(* Logix 5000 project; controller Hose_HP_Test_Rig_V1 vendor 1 type 14 code 149 rev 32.11; software revision 32.00; part 3 of 10 *)
(* tags used below, declared in another part *)
   DOOR_CLOSE_STS_STN1 : DINT;
   EXHS_OK_DEL_STN1 : TIMER;
   EXHS_VAL_OFF_CE_STN1 : BOOL;
   EXHS_VAL_OFF_TE_STN1 : BOOL;
   ONS26 : BOOL;
   ONS27 : BOOL;
   ONS43 : BOOL;
   ONS44 : BOOL;
   ONS45 : BOOL;
   ONS71 : BOOL;
   ONS72 : BOOL;
   ONS73 : BOOL;
   ONS74 : BOOL;
   ONS75 : BOOL;
   PASS_COUNTER_STN1 : COUNTER;
   PASS_COUNTER_STN2 : COUNTER;
   PASS_COUNTER_STN3 : COUNTER;
   PASS_COUNTER_STN4 : COUNTER;
   RST_TOP_NOT_DECLAMPED_STN1 : BOOL;
   RST_TOP_NOT_DECLAMPED_STN2 : BOOL;
   RST_TOP_NOT_DECLAMPED_STN3 : BOOL;
   RST_TOP_NOT_DECLAMPED_STN4 : BOOL;
   ABORT_STN1 : BOOL;
   ACT_DROP_STN1 : REAL;
   ACT_PR_STN1 : REAL;
   AUTO_DOOR_OPEN_BLK_STN1 : DA_SOL_RET_SEQ;
   AUTO_DOOR_OPEN_BLK_STN2 : DA_SOL_RET_SEQ;
   AUTO_DOOR_OPEN_BLK_STN3 : DA_SOL_RET_SEQ;
   AUTO_DOOR_OPEN_BLK_STN4 : DA_SOL_RET_SEQ;
   AUTO_DOOR_OPEN_ON : BOOL;
   AUTO_DOOR_OPEN_ON_STN2 : BOOL;
   AUTO_DOOR_OPEN_ON_STN3 : BOOL;
   AUTO_DOOR_OPEN_ON_STN4 : BOOL;
   AUTO_DOOR_OPEN_SEQ : DINT;
   AUTO_DOOR_OPEN_SEQ_STN2 : DINT;
   AUTO_DOOR_OPEN_SEQ_STN3 : DINT;
   AUTO_DOOR_OPEN_SEQ_STN4 : DINT;
   AUTO_TEST_ON_STN1 : BOOL;
   AUTO_TEST_ON_STN2 : BOOL;
   AUTO_TEST_ON_STN3 : BOOL;
   AUTO_TEST_ON_STN4 : BOOL;
   AUTO_TEST_OVER_STN1 : BOOL;
   AUTO_TEST_OVER_STN2 : BOOL;
   AUTO_TEST_OVER_STN3 : BOOL;
   AUTO_TEST_OVER_STN4 : BOOL;
   AUTO_TEST_SEL_STN1 : BOOL;
   AUTO_TEST_SEL_STN2 : BOOL;
   AUTO_TEST_SEL_STN3 : BOOL;
   AUTO_TEST_SEL_STN4 : BOOL;
   BOTTOM_CLAMP_AUTO_STN1 : BOOL;
   BOTTOM_CLAMP_BLK_STN1 : DA_SOL_FWD_SEQ;
   BOTTOM_CLAMP_OK_STN1 : BOOL;
   BOTTOM_CLAMP_PR_CHK : TIMER;
   BOTTOM_CLAMP_PS_STN1 : ALIAS FOR Local:1:I.Data.13;
   BOTTOM_CLAMP_PS_STN2 : ALIAS FOR Local:2:I.Data.2;
   BOTTOM_CLAMP_PS_STN3 : ALIAS FOR Local:2:I.Data.7;
   BOTTOM_CLAMP_PS_STN4 : ALIAS FOR Local:2:I.Data.12;
   BOTTOM_CLAMP_SEQ_STN1 : DINT;
   BOTTOM_CLAMP_SOL_STN1 : ALIAS FOR Local:1:O.Data.4;
   BOTTOM_DECLAMP_AUTO_STN1 : BOOL;
   BOTTOM_DECLAMP_SEQ_STN1 : DINT;
   BOTTOM_DECLMP_BLK_STN1 : DA_SOL_RET_SEQ;
   BOTTOM_NOT_CLAMPED_STN1 : BOOL;
   BOTTOM_NOT_DECLAMPED_STN1 : BOOL;
   CHECK_TRACE_STS_STN1 : BOOL;
   CLR_FAIL_ONS_STN1 : BOOL;
   CLR_ONS_STN1 : BOOL;
   COMP_FAULT_STN1 : BOOL;
   CONS_CALB_OFF_STN1 : BOOL;
   CONS_CALB_OFF_STN2 : BOOL;
   CONS_CALB_OFF_STN3 : BOOL;
   CONS_CALB_OFF_STN4 : BOOL;
   CONS_CALB_ON_STN1 : BOOL;
   CONS_STS_STN1 : DINT;
   CONS_TEST_ON : BOOL;
   CONSTRICTION_TEST_ON_STN1 : BOOL;
   CONSTRICTION_TEST_ON_STN2 : BOOL;
   CONSTRICTION_TEST_ON_STN3 : BOOL;
   CONSTRICTION_TEST_ON_STN4 : BOOL;
   DICH_STN1 : INT;
   DOOR_CLOSE_ABORT_STN1 : BOOL;
   DOOR_CLOSE_AUTO_STN1 : BOOL;
   DOOR_CLOSE_BLK_STN1 : DOOR_CLOSE;
   DOOR_CLOSE_OK_STN1 : BOOL;
   DOOR_CLOSE_RS_STN1 : ALIAS FOR Local:1:I.Data.11;
   DOOR_CLOSE_SEQ_STN1 : DA_SOL_FWD_SEQ;
   DOOR_NOT_CLOSED : BOOL;
   DOOR_NOT_OPEN_STN1 : BOOL;
   DOOR_NOT_OPEN_STN2 : BOOL;
   DOOR_NOT_OPEN_STN3 : BOOL;
   DOOR_NOT_OPEN_STN4 : BOOL;
   DOOR_OPEN_RS_STN1 : ALIAS FOR Local:1:I.Data.10;
   DOOR_OPEN_RS_STN2 : ALIAS FOR Local:1:I.Data.15;
   DOOR_OPEN_RS_STN3 : ALIAS FOR Local:2:I.Data.4;
   DOOR_OPEN_RS_STN4 : ALIAS FOR Local:2:I.Data.10;
   DROP_CHK_SEQ_STN1 : DROP_CHECK;
   DROP_NOK_STN1 : BOOL;
   DROP_OK_STN1 : BOOL;
   DUPLICATE_STN1 : BOOL;
   EC_STN1 : DINT;
   EC_STN2 : DINT;
   EC_STN3 : DINT;
   EC_STN4 : DINT;
   EXHAUST_SET_LIM : REAL;
   EXHS_OFF_BLK_STN1 : FILL_VAL_OFF;
   EXHS_VAL_HP_ON_STN1 : BOOL;
   EXHS_VAL_OFF_STN1 : BOOL;
   FAILED_STN1 : BOOL;
   FAILED_STN2 : BOOL;
   FAILED_STN3 : BOOL;
   FAILED_STN4 : BOOL;
   FAULTED_STN1 : BOOL;
   FAULTED_STN2 : BOOL;
   FAULTED_STN3 : BOOL;
   FAULTED_STN4 : BOOL;
   FILL_ACT_TIME_STN1 : REAL;
   FILL_CHK_STN1 : PR_CHECK;
   FILL_HIGH_STN1 : BOOL;
   FILL_HL_STN1 : REAL;
   FILL_LL_STN1 : REAL;
   FILL_LOW_STN1 : BOOL;
   FILL_SEQ_START_STN : SEQ_START_AND_FILL;
   FILL_SET_TIME : REAL;
   FILL_VAL_OFF_SEQ_STN1 : FILL_VAL_OFF;
   FLT_CLR_ONS_STN1 : BOOL;
   FLT_CLR_ONS_STN2 : BOOL;
   FLT_CLR_ONS_STN3 : BOOL;
   FLT_CLR_ONS_STN4 : BOOL;
   FLT_CODE_STN4 : DINT;
   HP_P2_STN1 : REAL;
   HP_STS_STN1 : DINT;
   HP_TEST_ON : BOOL;
   INCORRECT_STN1 : BOOL;
   INIT_STN1 : BOOL;
   LT_COMPLETED_STN1 : BOOL;
   LT_P1_STN1 : REAL;
   LT_POKEYOKE_STN1 : DINT;
   MSG_STN1 : DINT;
   MSG_STN2 : DINT;
   MSG_STN3 : DINT;
   MSG_STN4 : DINT;
   P2_STN1 : REAL;
   PASS_COUNT_RETEST : DINT;
   PASS_COUNT_RETEST_STN2 : DINT;
   PASS_COUNT_STN1 : DINT;
   PASS_COUNT_STN2 : DINT;
   PASS_COUNT_STN3 : DINT;
   PASS_COUNT_STN4 : DINT;
   PASS_COUNTER_RETEST : COUNTER;
   PASS_COUNTER_RETEST_STN2 : COUNTER;
   PASSED_STN1 : BOOL;
   PASSED_STN2 : BOOL;
   PASSED_STN3 : BOOL;
   PASSED_STN4 : BOOL;
   POKEYOKE_NOT_DONE : BOOL;
   PYOKE_LT_STN1 : BOOL;
   RETEST : BOOL;
   RST_EXHS_VAL_OFF_STN1 : BOOL;
   RST_SEQ_ON_STN1 : BOOL;
   RST_TEST_VAL_OFF_STN1 : BOOL;
   SCAN_OK_STN1 : BOOL;
   SCR_STS : DINT[6];
   SEQ_NO_STN1 : DINT;
   SEQ_NO_STN2 : DINT;
   SEQ_NO_STN3 : DINT;
   SEQ_NO_STN4 : DINT;
   SET_DROP : REAL;
   STAB_ACT_TIME_STN1 : REAL;
   STAB_CHK_STN1 : PR_CHECK;
   STAB_HIGH_STN1 : BOOL;
   STAB_LOW_STN1 : BOOL;
   STAB_SET_TIME : REAL;
   STAMP_BLK_STN1 : STAMP_SEQ;
   STAMP_BLK_STN2 : STAMP_SEQ;
   STAMP_BLK_STN3 : STAMP_SEQ;
   STAMP_BLK_STN4 : STAMP_SEQ;
   STAMP_FWD_OK_STN1 : BOOL;
   STAMP_FWD_OK_STN2 : BOOL;
   STAMP_FWD_OK_STN3 : BOOL;
   STAMP_FWD_OK_STN4 : BOOL;
   STAMP_NOT_FWD : BOOL;
   STAMP_NOT_FWD_STN2 : BOOL;
   STAMP_NOT_FWD_STN3 : BOOL;
   STAMP_NOT_FWD_STN4 : BOOL;
   STAMP_ON_STN1 : BOOL;
   STAMP_ON_STN2 : BOOL;
   STAMP_ON_STN3 : BOOL;
   STAMP_ON_STN4 : BOOL;
   STAMP_PS_STN1 : ALIAS FOR Local:1:I.Data.14;
   STAMP_PS_STN2 : ALIAS FOR Local:2:I.Data.3;
   STAMP_PS_STN3 : ALIAS FOR Local:2:I.Data.8;
   STAMP_PS_STN4 : ALIAS FOR Local:2:I.Data.13;
   STN1_ON : BOOL;
   STN1_TEST_STS : DINT;
   STN2_TEST_STS : DINT;
   STN3_TEST_STS : DINT;
   STN4_TEST_STS : DINT;
   STS_OP_STN1 : DINT;
   TEST_ACT_TIME_STN1 : REAL;
   TEST_ON_STN1 : BOOL;
   TEST_ON_STN2 : BOOL;
   TEST_ON_STN3 : BOOL;
   TEST_ON_STN4 : BOOL;
   TEST_OVER_DEL : TIMER;
   TEST_OVER_DEL_STN2 : TIMER;
   TEST_OVER_DEL_STN3 : TIMER;
   TEST_OVER_DEL_STN4 : TIMER;
   TEST_SET_TIME : REAL;
   TEST_STS_STN1 : DINT;
   TEST_STS_UPDATE_STN1 : TEST_TAIL_END;
   TEST_VAL_OFF_STN1 : BOOL;
   TEST_VAL_ON_STN1 : BOOL;
   TOP_CLAMP_AUTO_STN1 : BOOL;
   TOP_CLAMP_BLK_STN1 : DA_SOL_FWD_SEQ;
   TOP_CLAMP_OK_STN1 : BOOL;
   TOP_CLAMP_ON_SEQ_STN1 : DINT;
   TOP_CLAMP_PS_STN1 : ALIAS FOR Local:1:I.Data.12;
   TOP_CLAMP_PS_STN2 : ALIAS FOR Local:2:I.Data.1;
   TOP_CLAMP_PS_STN3 : ALIAS FOR Local:2:I.Data.6;
   TOP_CLAMP_PS_STN4 : ALIAS FOR Local:2:I.Data.11;
   TOP_DECLAMP_AUTO_STN1 : BOOL;
   TOP_DECLAMP_AUTO_STN2 : BOOL;
   TOP_DECLAMP_AUTO_STN3 : BOOL;
   TOP_DECLAMP_AUTO_STN4 : BOOL;
   TOP_DECLAMP_BLK_STN1 : TOP_DECLAMP;
   TOP_DECLAMP_BLK_STN2 : TOP_DECLAMP;
   TOP_DECLAMP_BLK_STN3 : TOP_DECLAMP;
   TOP_DECLAMP_BLK_STN4 : TOP_DECLAMP;
   TOP_DECLAMP_OK_STN1 : BOOL;
   TOP_DECLAMP_OK_STN2 : BOOL;
   TOP_DECLAMP_OK_STN3 : BOOL;
   TOP_DECLAMP_OK_STN4 : BOOL;
   TOP_NOT_CLAMPED_STN1 : BOOL;
   TOP_NOT_DECLAMPED_STN1 : BOOL;
   TOP_NOT_DECLAMPED_STN2 : BOOL;
   TOP_NOT_DECLAMPED_STN3 : BOOL;
   TOP_NOT_DECLAMPED_STN4 : BOOL;
   TRACE_ON_STN1 : BOOL;
   TS_STS_OP20A : DINT;
   TS_STS_STN1 : DINT;
   TS_STS_STN3 : DINT;
   TS_STS_STN4 : DINT;
(* MainProgram, continued *)

ROUTINE Auto_End_Stn1   (* ladder *)
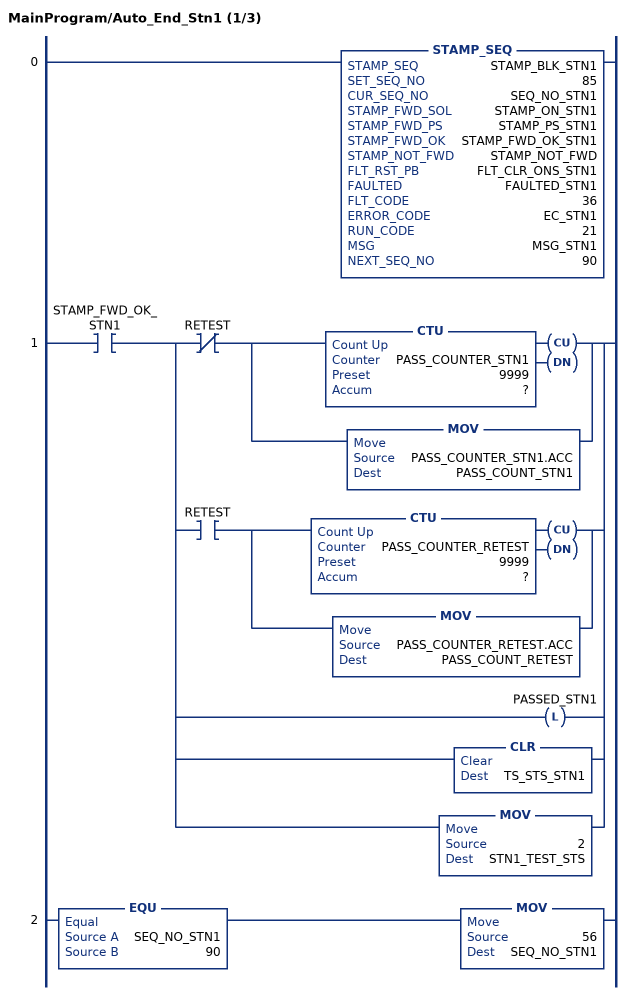
   0: STAMP_SEQ(STAMP_BLK_STN1,85,SEQ_NO_STN1,STAMP_ON_STN1,STAMP_PS_STN1,STAMP_FWD_OK_STN1,STAMP_NOT_FWD,FLT_CLR_ONS_STN1,FAULTED_STN1,36,EC_STN1,21,MSG_STN1,90);
   1: XIC(STAMP_FWD_OK_STN1)[XIO(RETEST) [CTU(PASS_COUNTER_STN1,?,?) ,MOV(PASS_COUNTER_STN1.ACC,PASS_COUNT_STN1) ] ,XIC(RETEST) [CTU(PASS_COUNTER_RETEST,?,?) ,MOV(PASS_COUNTER_RETEST.ACC,PASS_COUNT_RETEST) ] ,OTL(PASSED_STN1) ,CLR(TS_STS_STN1) ,MOV(2,STN1_TEST_STS) ];
   2: EQU(SEQ_NO_STN1,90)MOV(56,SEQ_NO_STN1);
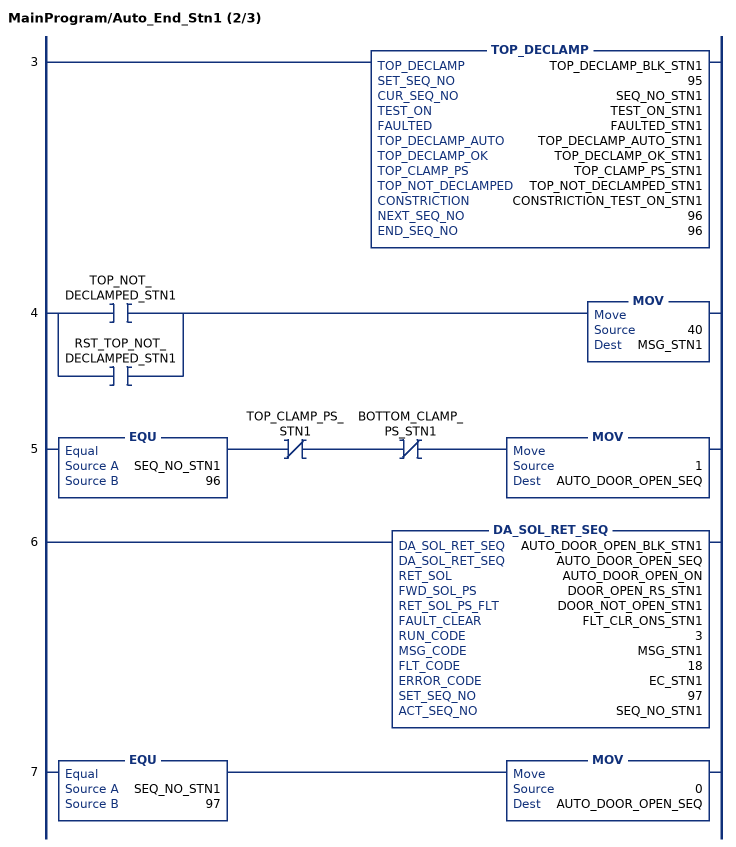
   3: TOP_DECLAMP(TOP_DECLAMP_BLK_STN1,95,SEQ_NO_STN1,TEST_ON_STN1,FAULTED_STN1,TOP_DECLAMP_AUTO_STN1,TOP_DECLAMP_OK_STN1,TOP_CLAMP_PS_STN1,TOP_NOT_DECLAMPED_STN1,CONSTRICTION_TEST_ON_STN1,96,96);
   4: [XIC(TOP_NOT_DECLAMPED_STN1) ,XIC(RST_TOP_NOT_DECLAMPED_STN1) ]MOV(40,MSG_STN1);
   5: EQU(SEQ_NO_STN1,96)XIO(TOP_CLAMP_PS_STN1)XIO(BOTTOM_CLAMP_PS_STN1)MOV(1,AUTO_DOOR_OPEN_SEQ);
   6: DA_SOL_RET_SEQ(AUTO_DOOR_OPEN_BLK_STN1,AUTO_DOOR_OPEN_SEQ,AUTO_DOOR_OPEN_ON,DOOR_OPEN_RS_STN1,DOOR_NOT_OPEN_STN1,FLT_CLR_ONS_STN1,3,MSG_STN1,18,EC_STN1,97,SEQ_NO_STN1);
   7: EQU(SEQ_NO_STN1,97)MOV(0,AUTO_DOOR_OPEN_SEQ);
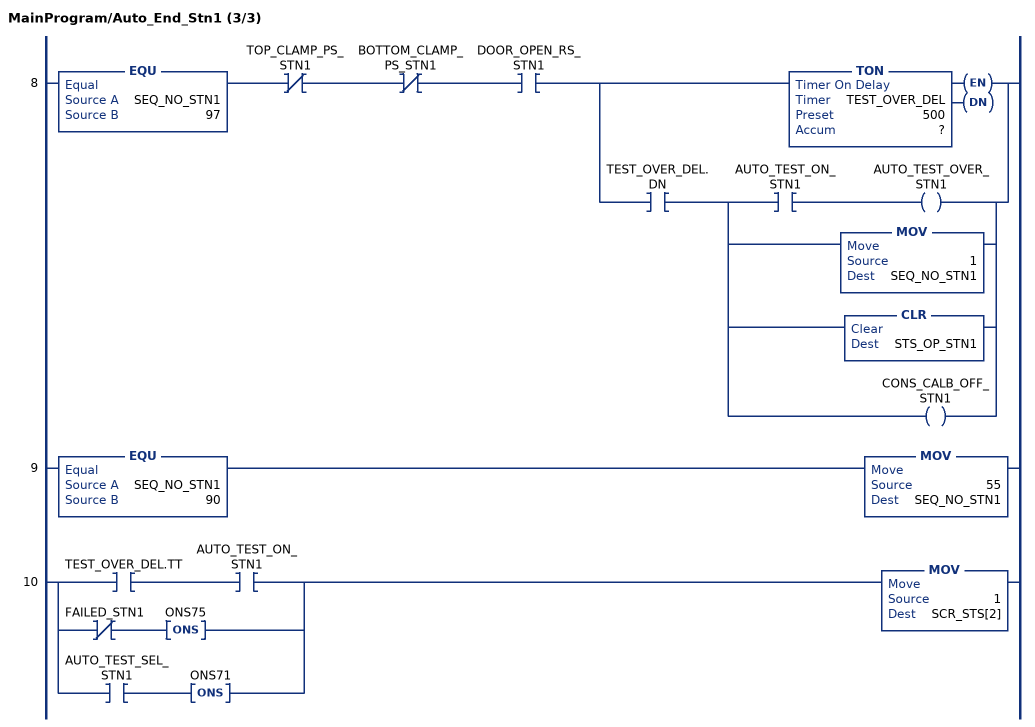
   8: EQU(SEQ_NO_STN1,97)XIO(TOP_CLAMP_PS_STN1)XIO(BOTTOM_CLAMP_PS_STN1)XIC(DOOR_OPEN_RS_STN1)[TON(TEST_OVER_DEL,?,?) ,XIC(TEST_OVER_DEL.DN) [[XIC(AUTO_TEST_ON_STN1) OTE(AUTO_TEST_OVER_STN1) ,MOV(1,SEQ_NO_STN1) ,CLR(STS_OP_STN1) ] ,OTE(CONS_CALB_OFF_STN1) ] ];
   9: EQU(SEQ_NO_STN1,90)MOV(55,SEQ_NO_STN1);
   10: [XIC(TEST_OVER_DEL.TT) XIC(AUTO_TEST_ON_STN1) ,XIO(FAILED_STN1) ONS(ONS75) ,XIC(AUTO_TEST_SEL_STN1) ONS(ONS71) ]MOV(1,SCR_STS[2]);
END_ROUTINE

ROUTINE Auto_End_Stn2   (* ladder *)
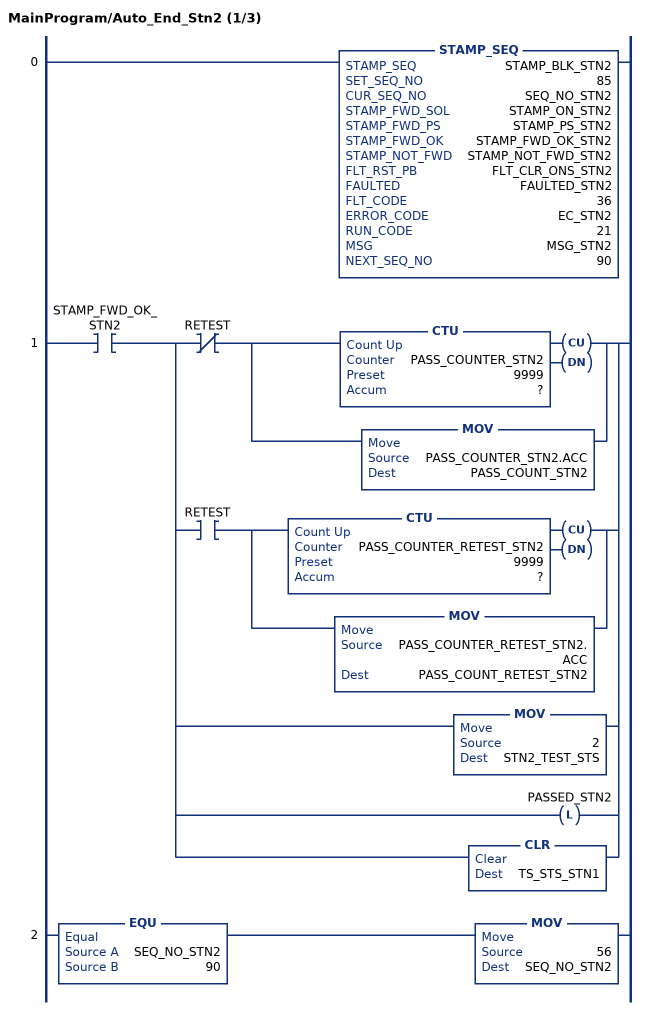
   0: STAMP_SEQ(STAMP_BLK_STN2,85,SEQ_NO_STN2,STAMP_ON_STN2,STAMP_PS_STN2,STAMP_FWD_OK_STN2,STAMP_NOT_FWD_STN2,FLT_CLR_ONS_STN2,FAULTED_STN2,36,EC_STN2,21,MSG_STN2,90);
   1: XIC(STAMP_FWD_OK_STN2)[XIO(RETEST) [CTU(PASS_COUNTER_STN2,?,?) ,MOV(PASS_COUNTER_STN2.ACC,PASS_COUNT_STN2) ] ,XIC(RETEST) [CTU(PASS_COUNTER_RETEST_STN2,?,?) ,MOV(PASS_COUNTER_RETEST_STN2.ACC,PASS_COUNT_RETEST_STN2) ] ,MOV(2,STN2_TEST_STS) ,OTL(PASSED_STN2) ,CLR(TS_STS_STN1) ];
   2: EQU(SEQ_NO_STN2,90)MOV(56,SEQ_NO_STN2);
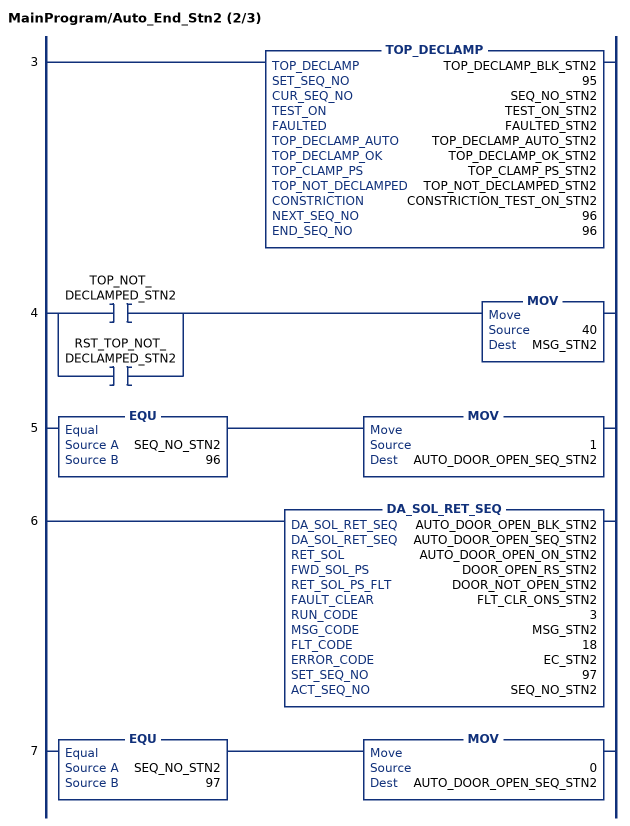
   3: TOP_DECLAMP(TOP_DECLAMP_BLK_STN2,95,SEQ_NO_STN2,TEST_ON_STN2,FAULTED_STN2,TOP_DECLAMP_AUTO_STN2,TOP_DECLAMP_OK_STN2,TOP_CLAMP_PS_STN2,TOP_NOT_DECLAMPED_STN2,CONSTRICTION_TEST_ON_STN2,96,96);
   4: [XIC(TOP_NOT_DECLAMPED_STN2) ,XIC(RST_TOP_NOT_DECLAMPED_STN2) ]MOV(40,MSG_STN2);
   5: EQU(SEQ_NO_STN2,96)MOV(1,AUTO_DOOR_OPEN_SEQ_STN2);
   6: DA_SOL_RET_SEQ(AUTO_DOOR_OPEN_BLK_STN2,AUTO_DOOR_OPEN_SEQ_STN2,AUTO_DOOR_OPEN_ON_STN2,DOOR_OPEN_RS_STN2,DOOR_NOT_OPEN_STN2,FLT_CLR_ONS_STN2,3,MSG_STN2,18,EC_STN2,97,SEQ_NO_STN2);
   7: EQU(SEQ_NO_STN2,97)MOV(0,AUTO_DOOR_OPEN_SEQ_STN2);
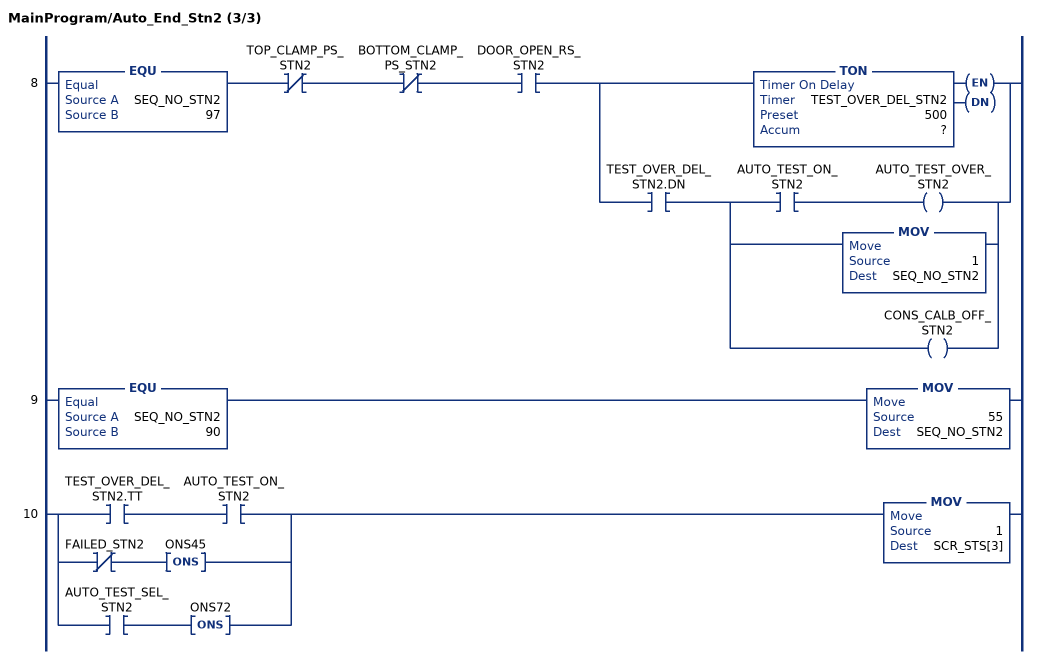
   8: EQU(SEQ_NO_STN2,97)XIO(TOP_CLAMP_PS_STN2)XIO(BOTTOM_CLAMP_PS_STN2)XIC(DOOR_OPEN_RS_STN2)[TON(TEST_OVER_DEL_STN2,?,?) ,XIC(TEST_OVER_DEL_STN2.DN) [XIC(AUTO_TEST_ON_STN2) OTE(AUTO_TEST_OVER_STN2) ,MOV(1,SEQ_NO_STN2) ,OTE(CONS_CALB_OFF_STN2) ] ];
   9: EQU(SEQ_NO_STN2,90)MOV(55,SEQ_NO_STN2);
   10: [XIC(TEST_OVER_DEL_STN2.TT) XIC(AUTO_TEST_ON_STN2) ,XIO(FAILED_STN2) ONS(ONS45) ,XIC(AUTO_TEST_SEL_STN2) ONS(ONS72) ]MOV(1,SCR_STS[3]);
END_ROUTINE

ROUTINE Auto_End_Stn3   (* ladder *)
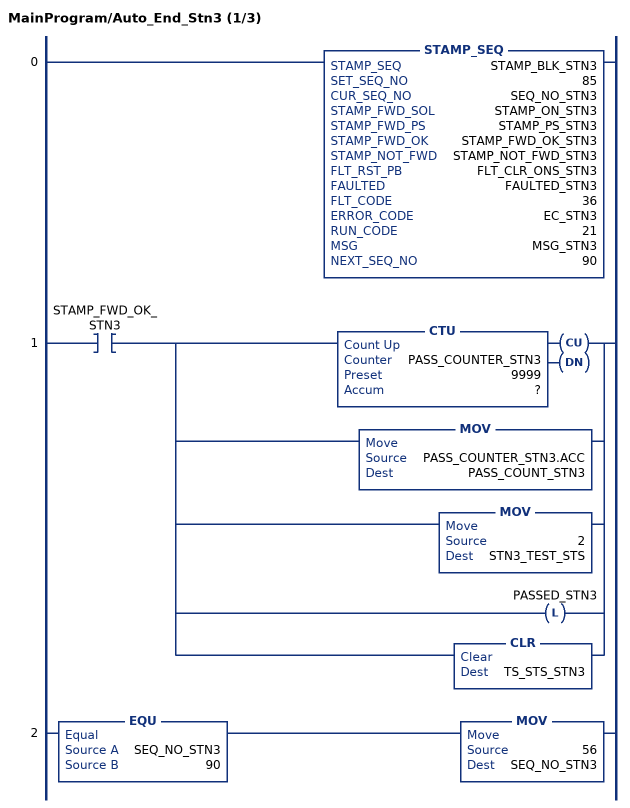
   0: STAMP_SEQ(STAMP_BLK_STN3,85,SEQ_NO_STN3,STAMP_ON_STN3,STAMP_PS_STN3,STAMP_FWD_OK_STN3,STAMP_NOT_FWD_STN3,FLT_CLR_ONS_STN3,FAULTED_STN3,36,EC_STN3,21,MSG_STN3,90);
   1: XIC(STAMP_FWD_OK_STN3)[CTU(PASS_COUNTER_STN3,?,?) ,MOV(PASS_COUNTER_STN3.ACC,PASS_COUNT_STN3) ,MOV(2,STN3_TEST_STS) ,OTL(PASSED_STN3) ,CLR(TS_STS_STN3) ];
   2: EQU(SEQ_NO_STN3,90)MOV(56,SEQ_NO_STN3);
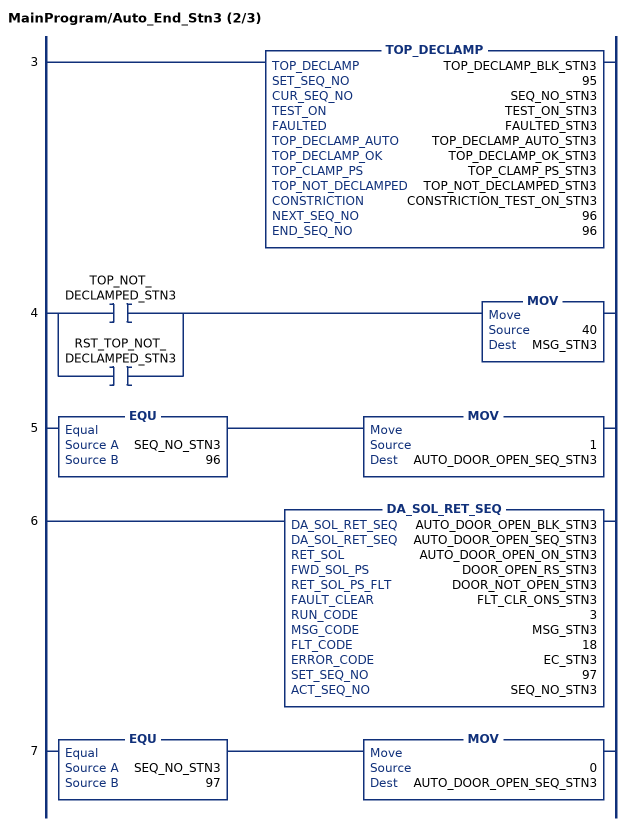
   3: TOP_DECLAMP(TOP_DECLAMP_BLK_STN3,95,SEQ_NO_STN3,TEST_ON_STN3,FAULTED_STN3,TOP_DECLAMP_AUTO_STN3,TOP_DECLAMP_OK_STN3,TOP_CLAMP_PS_STN3,TOP_NOT_DECLAMPED_STN3,CONSTRICTION_TEST_ON_STN3,96,96);
   4: [XIC(TOP_NOT_DECLAMPED_STN3) ,XIC(RST_TOP_NOT_DECLAMPED_STN3) ]MOV(40,MSG_STN3);
   5: EQU(SEQ_NO_STN3,96)MOV(1,AUTO_DOOR_OPEN_SEQ_STN3);
   6: DA_SOL_RET_SEQ(AUTO_DOOR_OPEN_BLK_STN3,AUTO_DOOR_OPEN_SEQ_STN3,AUTO_DOOR_OPEN_ON_STN3,DOOR_OPEN_RS_STN3,DOOR_NOT_OPEN_STN3,FLT_CLR_ONS_STN3,3,MSG_STN3,18,EC_STN3,97,SEQ_NO_STN3);
   7: EQU(SEQ_NO_STN3,97)MOV(0,AUTO_DOOR_OPEN_SEQ_STN3);
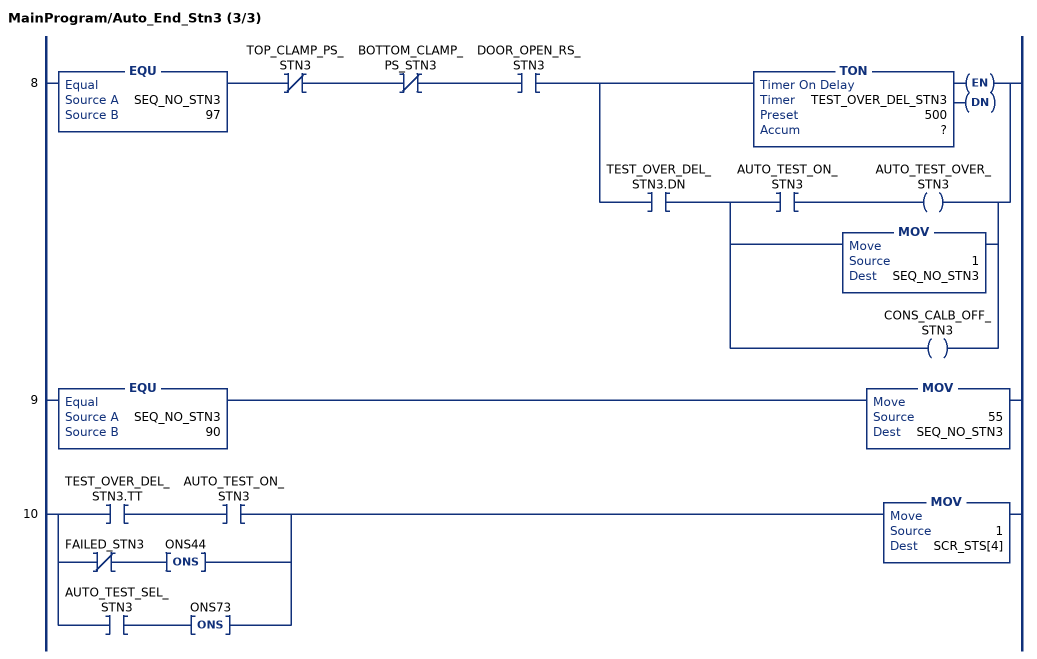
   8: EQU(SEQ_NO_STN3,97)XIO(TOP_CLAMP_PS_STN3)XIO(BOTTOM_CLAMP_PS_STN3)XIC(DOOR_OPEN_RS_STN3)[TON(TEST_OVER_DEL_STN3,?,?) ,XIC(TEST_OVER_DEL_STN3.DN) [XIC(AUTO_TEST_ON_STN3) OTE(AUTO_TEST_OVER_STN3) ,MOV(1,SEQ_NO_STN3) ,OTE(CONS_CALB_OFF_STN3) ] ];
   9: EQU(SEQ_NO_STN3,90)MOV(55,SEQ_NO_STN3);
   10: [XIC(TEST_OVER_DEL_STN3.TT) XIC(AUTO_TEST_ON_STN3) ,XIO(FAILED_STN3) ONS(ONS44) ,XIC(AUTO_TEST_SEL_STN3) ONS(ONS73) ]MOV(1,SCR_STS[4]);
END_ROUTINE

ROUTINE Auto_End_Stn4   (* ladder *)
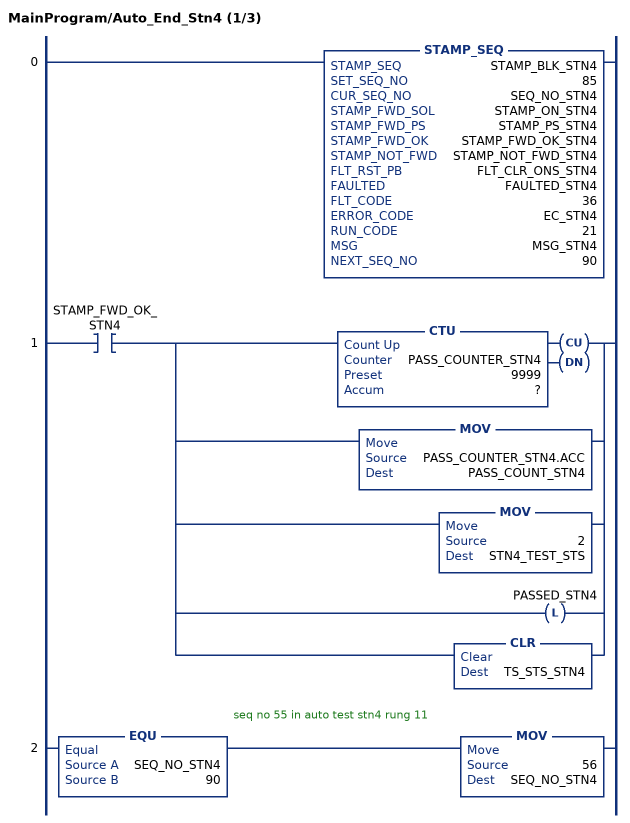
   0: STAMP_SEQ(STAMP_BLK_STN4,85,SEQ_NO_STN4,STAMP_ON_STN4,STAMP_PS_STN4,STAMP_FWD_OK_STN4,STAMP_NOT_FWD_STN4,FLT_CLR_ONS_STN4,FAULTED_STN4,36,EC_STN4,21,MSG_STN4,90);
   1: XIC(STAMP_FWD_OK_STN4)[CTU(PASS_COUNTER_STN4,?,?) ,MOV(PASS_COUNTER_STN4.ACC,PASS_COUNT_STN4) ,MOV(2,STN4_TEST_STS) ,OTL(PASSED_STN4) ,CLR(TS_STS_STN4) ];
   // seq no 55 in auto test stn4 rung 11
   2: EQU(SEQ_NO_STN4,90)MOV(56,SEQ_NO_STN4);
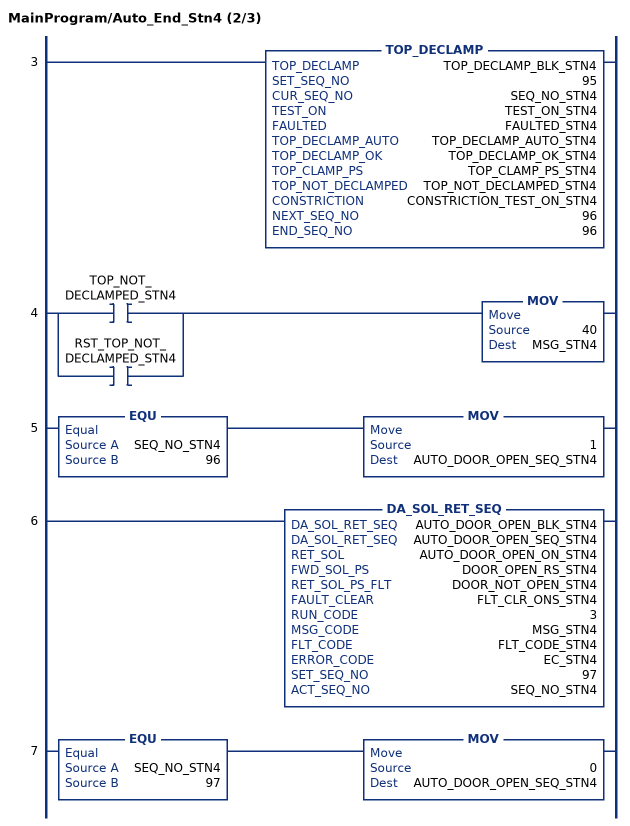
   3: TOP_DECLAMP(TOP_DECLAMP_BLK_STN4,95,SEQ_NO_STN4,TEST_ON_STN4,FAULTED_STN4,TOP_DECLAMP_AUTO_STN4,TOP_DECLAMP_OK_STN4,TOP_CLAMP_PS_STN4,TOP_NOT_DECLAMPED_STN4,CONSTRICTION_TEST_ON_STN4,96,96);
   4: [XIC(TOP_NOT_DECLAMPED_STN4) ,XIC(RST_TOP_NOT_DECLAMPED_STN4) ]MOV(40,MSG_STN4);
   5: EQU(SEQ_NO_STN4,96)MOV(1,AUTO_DOOR_OPEN_SEQ_STN4);
   6: DA_SOL_RET_SEQ(AUTO_DOOR_OPEN_BLK_STN4,AUTO_DOOR_OPEN_SEQ_STN4,AUTO_DOOR_OPEN_ON_STN4,DOOR_OPEN_RS_STN4,DOOR_NOT_OPEN_STN4,FLT_CLR_ONS_STN4,3,MSG_STN4,FLT_CODE_STN4,EC_STN4,97,SEQ_NO_STN4);
   7: EQU(SEQ_NO_STN4,97)MOV(0,AUTO_DOOR_OPEN_SEQ_STN4);
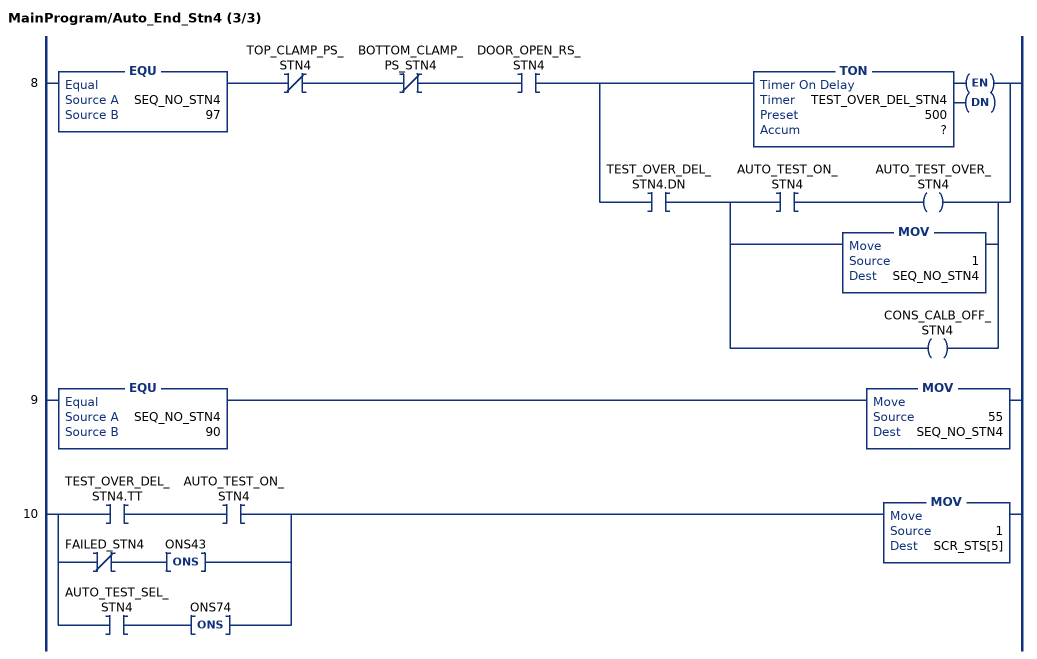
   8: EQU(SEQ_NO_STN4,97)XIO(TOP_CLAMP_PS_STN4)XIO(BOTTOM_CLAMP_PS_STN4)XIC(DOOR_OPEN_RS_STN4)[TON(TEST_OVER_DEL_STN4,?,?) ,XIC(TEST_OVER_DEL_STN4.DN) [XIC(AUTO_TEST_ON_STN4) OTE(AUTO_TEST_OVER_STN4) ,MOV(1,SEQ_NO_STN4) ,OTE(CONS_CALB_OFF_STN4) ] ];
   9: EQU(SEQ_NO_STN4,90)MOV(55,SEQ_NO_STN4);
   10: [XIC(TEST_OVER_DEL_STN4.TT) XIC(AUTO_TEST_ON_STN4) ,XIO(FAILED_STN4) ONS(ONS43) ,XIC(AUTO_TEST_SEL_STN4) ONS(ONS74) ]MOV(1,SCR_STS[5]);
END_ROUTINE

ROUTINE Auto_Test_Stn1   (* ladder *)
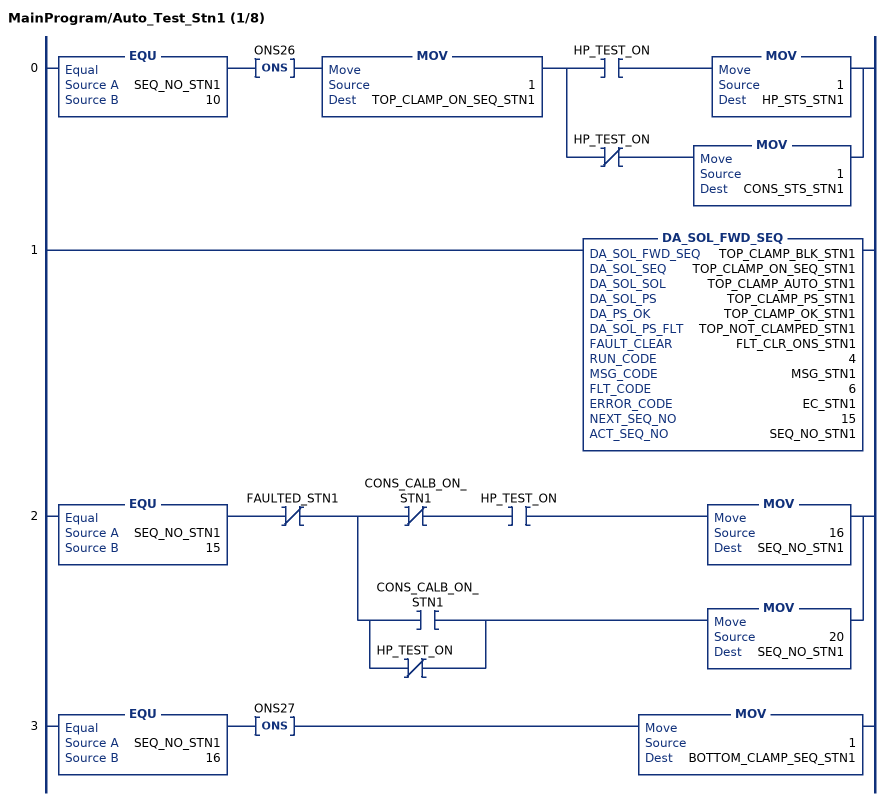
   0: EQU(SEQ_NO_STN1,10)ONS(ONS26)MOV(1,TOP_CLAMP_ON_SEQ_STN1)[XIC(HP_TEST_ON) MOV(1,HP_STS_STN1) ,XIO(HP_TEST_ON) MOV(1,CONS_STS_STN1) ];
   1: DA_SOL_FWD_SEQ(TOP_CLAMP_BLK_STN1,TOP_CLAMP_ON_SEQ_STN1,TOP_CLAMP_AUTO_STN1,TOP_CLAMP_PS_STN1,TOP_CLAMP_OK_STN1,TOP_NOT_CLAMPED_STN1,FLT_CLR_ONS_STN1,4,MSG_STN1,6,EC_STN1,15,SEQ_NO_STN1);
   2: EQU(SEQ_NO_STN1,15)XIO(FAULTED_STN1)[XIO(CONS_CALB_ON_STN1) XIC(HP_TEST_ON) MOV(16,SEQ_NO_STN1) ,[XIC(CONS_CALB_ON_STN1) ,XIO(HP_TEST_ON) ] MOV(20,SEQ_NO_STN1) ];
   3: EQU(SEQ_NO_STN1,16)ONS(ONS27)MOV(1,BOTTOM_CLAMP_SEQ_STN1);
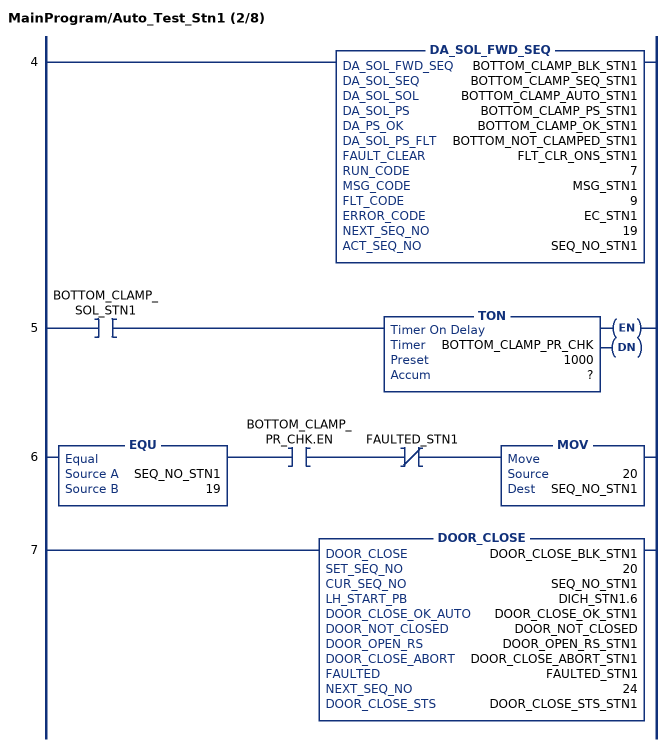
   4: DA_SOL_FWD_SEQ(BOTTOM_CLAMP_BLK_STN1,BOTTOM_CLAMP_SEQ_STN1,BOTTOM_CLAMP_AUTO_STN1,BOTTOM_CLAMP_PS_STN1,BOTTOM_CLAMP_OK_STN1,BOTTOM_NOT_CLAMPED_STN1,FLT_CLR_ONS_STN1,7,MSG_STN1,9,EC_STN1,19,SEQ_NO_STN1);
   5: XIC(BOTTOM_CLAMP_SOL_STN1)TON(BOTTOM_CLAMP_PR_CHK,?,?);
   6: EQU(SEQ_NO_STN1,19)XIC(BOTTOM_CLAMP_PR_CHK.EN)XIO(FAULTED_STN1)MOV(20,SEQ_NO_STN1);
   7: DOOR_CLOSE(DOOR_CLOSE_BLK_STN1,20,SEQ_NO_STN1,DICH_STN1.6,DOOR_CLOSE_OK_STN1,DOOR_NOT_CLOSED,DOOR_OPEN_RS_STN1,DOOR_CLOSE_ABORT_STN1,FAULTED_STN1,24,DOOR_CLOSE_STS_STN1);
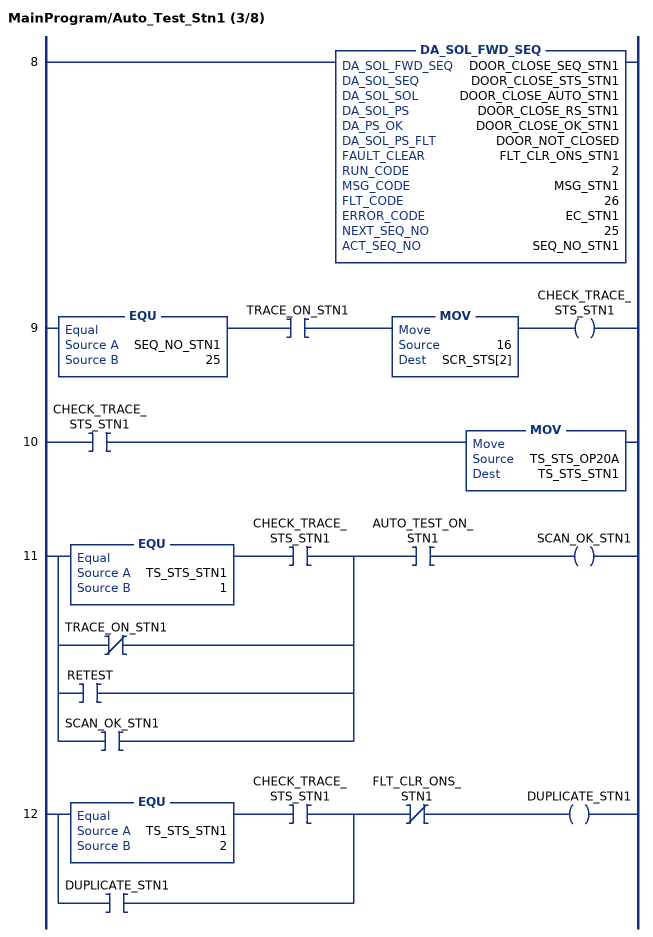
   8: DA_SOL_FWD_SEQ(DOOR_CLOSE_SEQ_STN1,DOOR_CLOSE_STS_STN1,DOOR_CLOSE_AUTO_STN1,DOOR_CLOSE_RS_STN1,DOOR_CLOSE_OK_STN1,DOOR_NOT_CLOSED,FLT_CLR_ONS_STN1,2,MSG_STN1,26,EC_STN1,25,SEQ_NO_STN1);
   9: EQU(SEQ_NO_STN1,25)XIC(TRACE_ON_STN1)MOV(16,SCR_STS[2])OTE(CHECK_TRACE_STS_STN1);
   10: XIC(CHECK_TRACE_STS_STN1)MOV(TS_STS_OP20A,TS_STS_STN1);
   11: [[EQU(TS_STS_STN1,1) XIC(CHECK_TRACE_STS_STN1) ,XIO(TRACE_ON_STN1) ,XIC(RETEST) ] ,XIC(SCAN_OK_STN1) ]XIC(AUTO_TEST_ON_STN1)OTE(SCAN_OK_STN1);
   12: [EQU(TS_STS_STN1,2) XIC(CHECK_TRACE_STS_STN1) ,XIC(DUPLICATE_STN1) ]XIO(FLT_CLR_ONS_STN1)OTE(DUPLICATE_STN1);
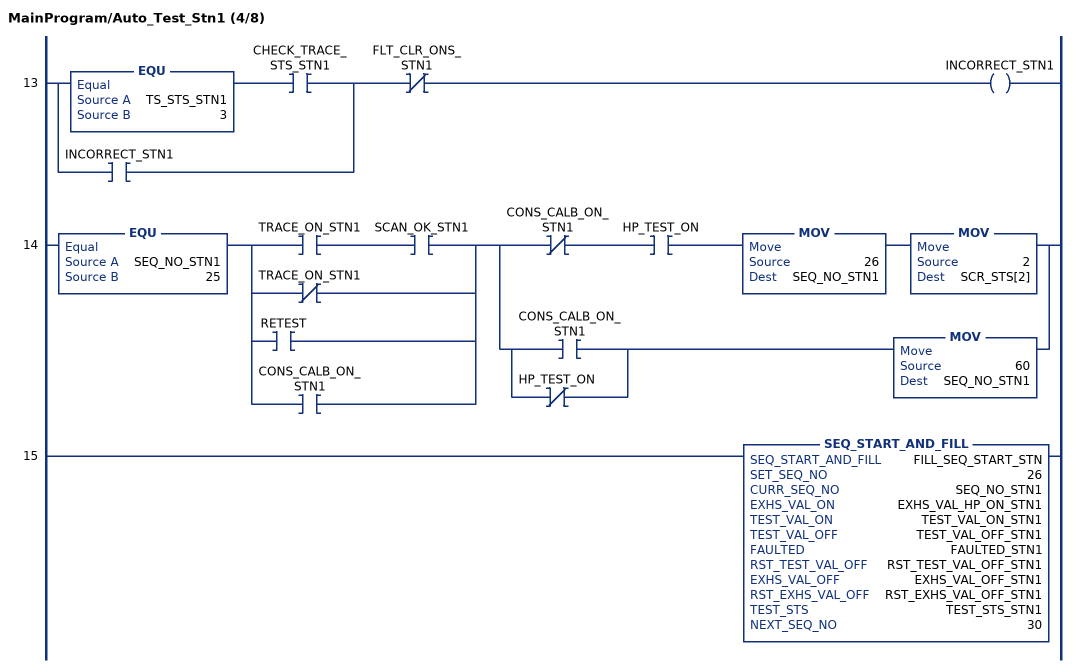
   13: [EQU(TS_STS_STN1,3) XIC(CHECK_TRACE_STS_STN1) ,XIC(INCORRECT_STN1) ]XIO(FLT_CLR_ONS_STN1)OTE(INCORRECT_STN1);
   14: EQU(SEQ_NO_STN1,25)[XIC(TRACE_ON_STN1) XIC(SCAN_OK_STN1) ,XIO(TRACE_ON_STN1) ,XIC(RETEST) ,XIC(CONS_CALB_ON_STN1) ][XIO(CONS_CALB_ON_STN1) XIC(HP_TEST_ON) MOV(26,SEQ_NO_STN1) MOV(2,SCR_STS[2]) ,[XIC(CONS_CALB_ON_STN1) ,XIO(HP_TEST_ON) ] MOV(60,SEQ_NO_STN1) ];
   15: SEQ_START_AND_FILL(FILL_SEQ_START_STN,26,SEQ_NO_STN1,EXHS_VAL_HP_ON_STN1,TEST_VAL_ON_STN1,TEST_VAL_OFF_STN1,FAULTED_STN1,RST_TEST_VAL_OFF_STN1,EXHS_VAL_OFF_STN1,RST_EXHS_VAL_OFF_STN1,TEST_STS_STN1,30);
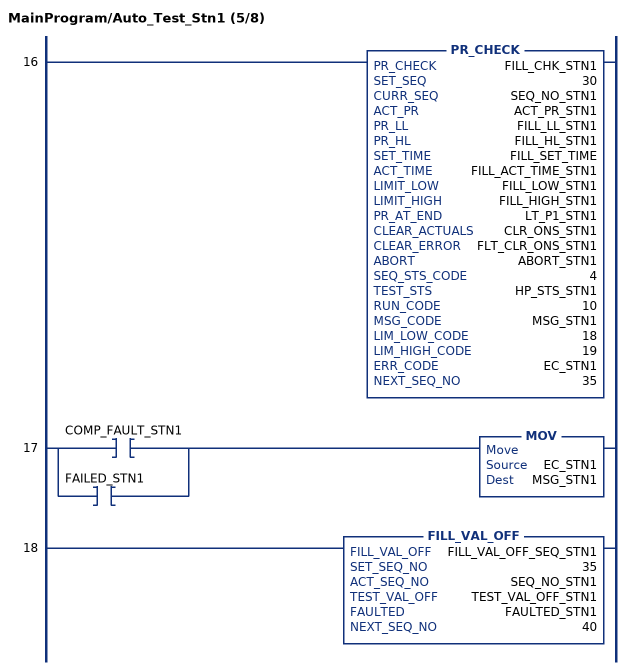
   16: PR_CHECK(FILL_CHK_STN1,30,SEQ_NO_STN1,ACT_PR_STN1,FILL_LL_STN1,FILL_HL_STN1,FILL_SET_TIME,FILL_ACT_TIME_STN1,FILL_LOW_STN1,FILL_HIGH_STN1,LT_P1_STN1,CLR_ONS_STN1,FLT_CLR_ONS_STN1,ABORT_STN1,4,HP_STS_STN1,10,MSG_STN1,18,19,EC_STN1,35);
   17: [XIC(COMP_FAULT_STN1) ,XIC(FAILED_STN1) ]MOV(EC_STN1,MSG_STN1);
   18: FILL_VAL_OFF(FILL_VAL_OFF_SEQ_STN1,35,SEQ_NO_STN1,TEST_VAL_OFF_STN1,FAULTED_STN1,40);
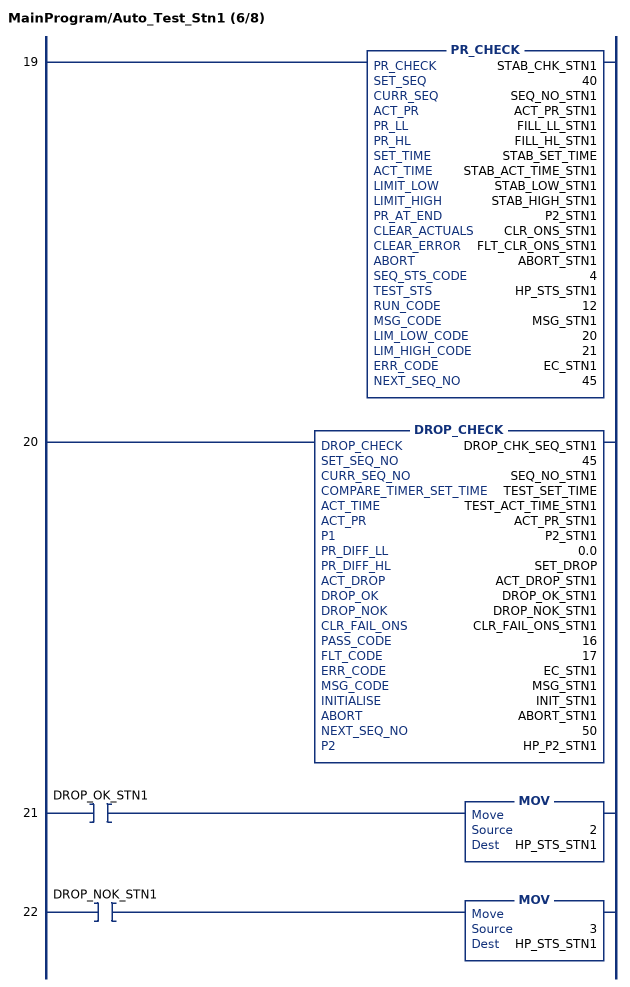
   19: PR_CHECK(STAB_CHK_STN1,40,SEQ_NO_STN1,ACT_PR_STN1,FILL_LL_STN1,FILL_HL_STN1,STAB_SET_TIME,STAB_ACT_TIME_STN1,STAB_LOW_STN1,STAB_HIGH_STN1,P2_STN1,CLR_ONS_STN1,FLT_CLR_ONS_STN1,ABORT_STN1,4,HP_STS_STN1,12,MSG_STN1,20,21,EC_STN1,45);
   20: DROP_CHECK(DROP_CHK_SEQ_STN1,45,SEQ_NO_STN1,TEST_SET_TIME,TEST_ACT_TIME_STN1,ACT_PR_STN1,P2_STN1,0.0,SET_DROP,ACT_DROP_STN1,DROP_OK_STN1,DROP_NOK_STN1,CLR_FAIL_ONS_STN1,16,17,EC_STN1,MSG_STN1,INIT_STN1,ABORT_STN1,50,HP_P2_STN1);
   21: XIC(DROP_OK_STN1)MOV(2,HP_STS_STN1);
   22: XIC(DROP_NOK_STN1)MOV(3,HP_STS_STN1);
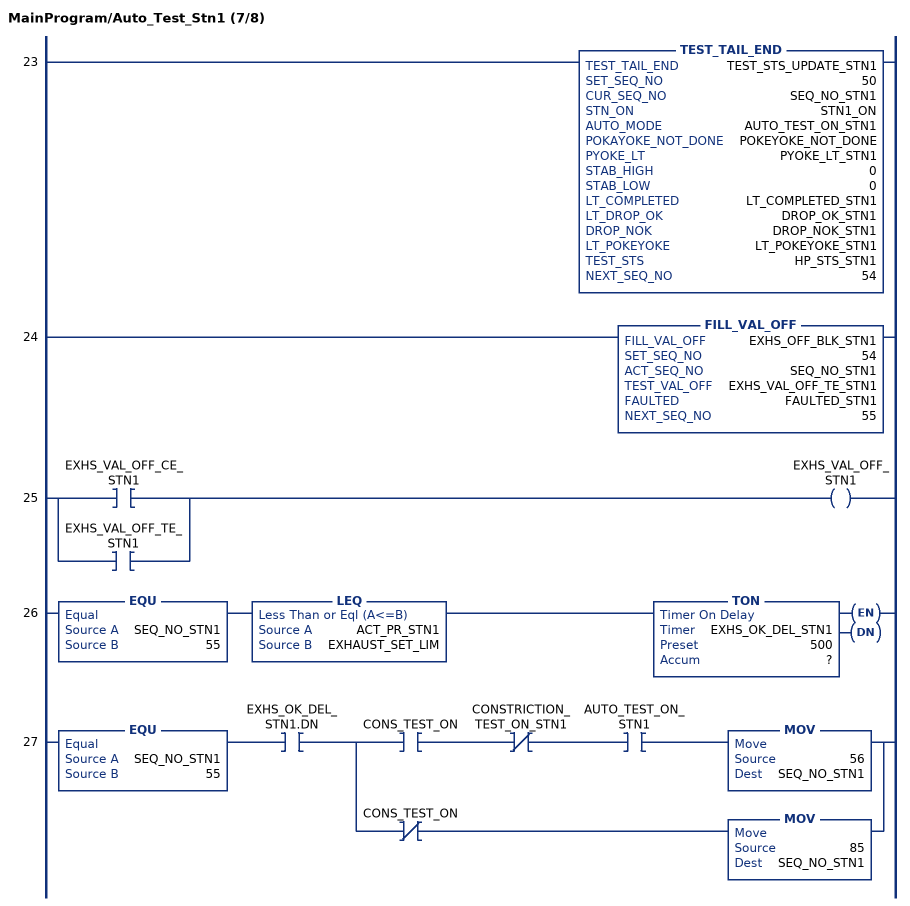
   23: TEST_TAIL_END(TEST_STS_UPDATE_STN1,50,SEQ_NO_STN1,STN1_ON,AUTO_TEST_ON_STN1,POKEYOKE_NOT_DONE,PYOKE_LT_STN1,0,0,LT_COMPLETED_STN1,DROP_OK_STN1,DROP_NOK_STN1,LT_POKEYOKE_STN1,HP_STS_STN1,54);
   24: FILL_VAL_OFF(EXHS_OFF_BLK_STN1,54,SEQ_NO_STN1,EXHS_VAL_OFF_TE_STN1,FAULTED_STN1,55);
   25: [XIC(EXHS_VAL_OFF_CE_STN1) ,XIC(EXHS_VAL_OFF_TE_STN1) ]OTE(EXHS_VAL_OFF_STN1);
   26: EQU(SEQ_NO_STN1,55)LEQ(ACT_PR_STN1,EXHAUST_SET_LIM)TON(EXHS_OK_DEL_STN1,?,?);
   27: EQU(SEQ_NO_STN1,55)XIC(EXHS_OK_DEL_STN1.DN)[XIC(CONS_TEST_ON) XIO(CONSTRICTION_TEST_ON_STN1) XIC(AUTO_TEST_ON_STN1) MOV(56,SEQ_NO_STN1) ,XIO(CONS_TEST_ON) MOV(85,SEQ_NO_STN1) ];
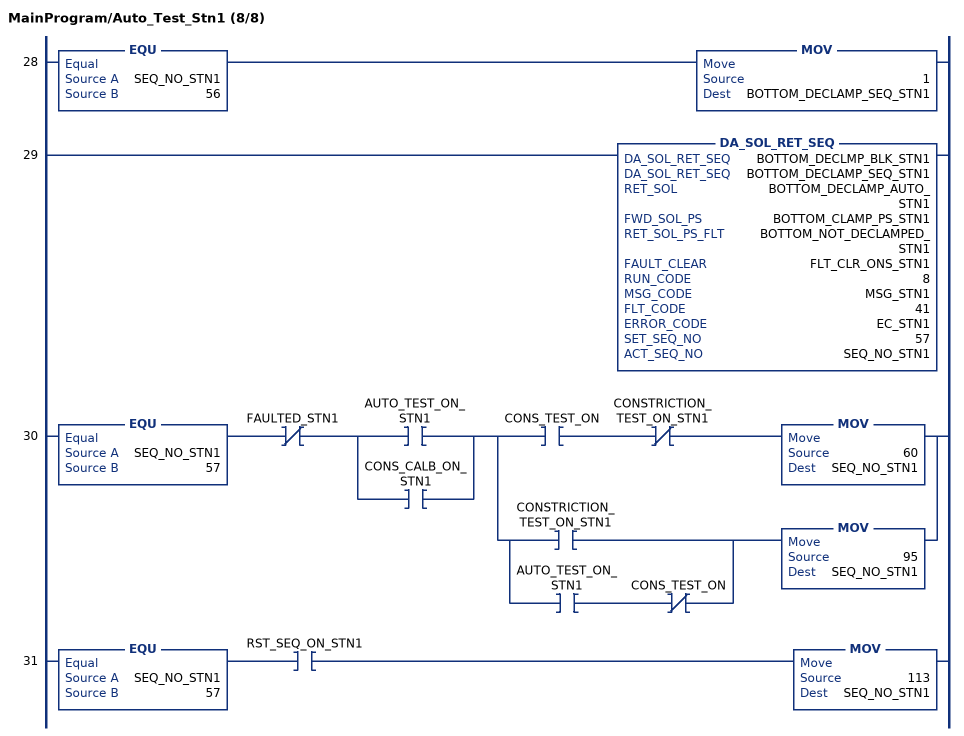
   28: EQU(SEQ_NO_STN1,56)MOV(1,BOTTOM_DECLAMP_SEQ_STN1);
   29: DA_SOL_RET_SEQ(BOTTOM_DECLMP_BLK_STN1,BOTTOM_DECLAMP_SEQ_STN1,BOTTOM_DECLAMP_AUTO_STN1,BOTTOM_CLAMP_PS_STN1,BOTTOM_NOT_DECLAMPED_STN1,FLT_CLR_ONS_STN1,8,MSG_STN1,41,EC_STN1,57,SEQ_NO_STN1);
   30: EQU(SEQ_NO_STN1,57)XIO(FAULTED_STN1)[XIC(AUTO_TEST_ON_STN1) ,XIC(CONS_CALB_ON_STN1) ][XIC(CONS_TEST_ON) XIO(CONSTRICTION_TEST_ON_STN1) MOV(60,SEQ_NO_STN1) ,[XIC(CONSTRICTION_TEST_ON_STN1) ,XIC(AUTO_TEST_ON_STN1) XIO(CONS_TEST_ON) ] MOV(95,SEQ_NO_STN1) ];
   31: EQU(SEQ_NO_STN1,57)XIC(RST_SEQ_ON_STN1)MOV(113,SEQ_NO_STN1);
END_ROUTINE
